// TIA Portal V17 export
// export: Created 2025-06-25T13:13:16.3780709Z, ExportSetting WithDefaults, DisplayName Totally Integrated Automation Portal, DisplayVersion V17 Update 8, DisplayName TIA Portal Openness, DisplayVersion V17 Update 8, DisplayName TIA Portal Version Control Interface, DisplayVersion V17, DisplayName STEP 7 Professional, DisplayVersion V17 Update 8, DisplayName STEP 7 Safety, DisplayVersion V17 Update 6, DisplayName WinCC Advanced, DisplayVersion V17 Update 8
FUNCTION "SaturationPressure" : Void   // FC28, FBD
{ S7_Optimized_Access := 'TRUE' }
VERSION : 0.1
// stored: AutoNumber true, IsIECCheckEnabled false, SetENOAutomatically false, UDAEnableTagReadback false
   VAR_INPUT
      Temperature : Real;
   END_VAR
   VAR_OUTPUT
      Pressure : Real;
   END_VAR
   VAR_TEMP
      CalcPressure : Real;
   END_VAR
   VAR_TEMP   // added for the SCL form of the ladder/FBD networks
      _w1 : Bool;
   END_VAR
BEGIN

REGION Network 1
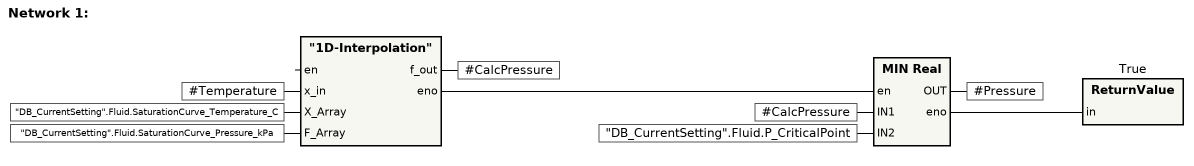
   "1D-Interpolation"(x_in := #Temperature,
                      X_Array := "DB_CurrentSetting".Fluid.SaturationCurve_Temperature_C,
                      F_Array := "DB_CurrentSetting".Fluid.SaturationCurve_Pressure_kPa,
                      f_out => #CalcPressure,
                      ENO => #_w1);
   IF #_w1 THEN
       #Pressure := MIN(IN1 := #CalcPressure, IN2 := "DB_CurrentSetting".Fluid.P_CriticalPoint);
       ENO := True;
       RETURN;
   END_IF;
END_REGION
END_FUNCTION
